FUNCTION_BLOCK FB_UnderfloorHeatingSystem EXTENDS FB_SystemContinous
VAR_INPUT
	bHeatingModeAutomatic : BOOL; //control mode: 0 = heating mode, 1 = cooling mode
	stAmbientState : ST_AmbientState;
END_VAR
VAR_OUTPUT
END_VAR
VAR
	{attribute 'OPC.UA.DA' := '1'}
	localSetParameters : ST_UnderfloorHeatingSetParameters;

	//default parameters
	localDefaultParameters : ST_UnderfloorHeatingDefaultParameters;	
	
	//pumps
	stPU425DefaultParameters : ST_PumpGrundfosMagna3DefaultParameters;
	PU425 : FB_PumpGrundfosMagna3 := (ST_DefaultParameters := stPU425DefaultParameters);	
	
	//valves
	stSV423DefaultParameters : ST_DiscreteValveDefaultParameters := (nFeedback := 3);
	stSV424DefaultParameters : ST_DiscreteValveDefaultParameters := (nFeedback := 3);
	stRV425DefaultParameters : ST_MixingValveDefaultParameters := (bFeedbackSignal := FALSE, tTaskCycleTime := GlobalVariables.tTaskCycleTime_MAIN, tCtrlCycleTime := GlobalVariables.tCtrlCycleTime_MAIN);	
	
	SV423 : FB_DiscreteValve := (ST_DefaultParameters := stSV423DefaultParameters); 
	SV424 : FB_DiscreteValve := (ST_DefaultParameters := stSV424DefaultParameters);
	RV425 : FB_MixingValve := (ST_DefaultParameters := stRV425DefaultParameters);
	
	//internal variables
	bHeatingMode 			: BOOL;
	bSetStatusOn_PU425 		: BOOL;
	bSetStatusOn_SV423		: BOOL;
	bSetStatusOn_SV424		: BOOL;
	bSetStatusOn_RV425 		: BOOL;
	fSetPoint_Internal 		: REAL;
	nControlMode_RV425 		: E_MixingValveControlMode; 	
	
	//characteristic curves and controllers
	CharacteristicCurve 			: FB_CTRL_FLOW_TEMP_SETPOINT_GEN;
	CharacteristicCurve_Parameters	: ST_CTRL_FLOW_TEMP_SETPOINT_GEN_PARAMS;
	
	//triggers
	SwitchToHeating : R_TRIG;
	SwitchToCooling : F_TRIG;
	bFinishedSwitchMode : BOOL := TRUE;
END_VAR

//check if heating mode has switched
SelectUnderfloorHeatingControlMode();
ControlUnderfloorHeating();
fSetPointAutomatic := fSetPoint_Internal;
SwitchToHeating(CLK := bHeatingMode);
SwitchToCooling(CLK := bHeatingMode);

//MAIN must be called before SwitchMode to prevent pump signal chattering (signal is written after SwitchMode function), SwitchMode may only be called if system is on
MAIN();

//disrupt calling SystemFlowControl via MAIN() when mode is switched and call SwitchMode()
IF ((SwitchToHeating.Q OR SwitchToCooling.Q) OR NOT bFinishedSwitchMode) AND bSetStatusOn THEN
	SwitchMode(bSwitchToHeating := bHeatingMode,
		bFinishedSwitchMode => bFinishedSwitchMode);
END_IF;

//pumps
PU425.GetState_Profibus();
PU425(bSetStatusOnAutomatic := bSetStatusOn_PU425,
	fSetPointAutomatic := 80,
	bAlgorithmPermission := bAlgorithmPermission,
	nControlModeAutomatic := 0);
PU425.SetState_Profibus();

//valves in thermal networks
RV425.GetState_AI();
RV425(bSetStatusOnAutomatic := bSetStatusOn_RV425,
	fSetPointAutomatic := fSetPoint_Internal,
	bAlgorithmPermission := bAlgorithmPermission,
	fTemperatureExternal := PU425.fTemperatureInternal,
	nControlModeAutomatic := nControlMode_RV425);
RV425.SetState_AO();

SV423.GetState_BI();
SV423(bSetStatusOnAutomatic := bSetStatusOn_SV423,
	bAlgorithmPermission := bAlgorithmPermission);
SV423.SetState_BO();

SV424.GetState_BI();
SV424(bSetStatusOnAutomatic := bSetStatusOn_SV423,
	bAlgorithmPermission := bAlgorithmPermission);
SV424.SetState_BO();

METHOD PROTECTED  CheckError : BOOL
VAR_INPUT
END_VAR
VAR_OUTPUT
	bError : BOOL;
END_VAR
VAR
END_VAR
//check pumps for errors
bError :=  PU425.bError;
END_METHOD

METHOD PRIVATE ControlUnderfloorHeating : BOOL
VAR_INPUT
END_VAR
VAR
END_VAR
CharacteristicCurve_Parameters.fAmbientTempMax := localDefaultParameters.aLimitsAmbientTemperature[2];
CharacteristicCurve_Parameters.fAmbientTempMin := localDefaultParameters.aLimitsAmbientTemperature[1];
CharacteristicCurve_Parameters.fForeRunTempMax := localDefaultParameters.aLimitsFeedTemperature[1];
CharacteristicCurve_Parameters.fForeRunTempMin := localDefaultParameters.aLimitsFeedTemperature[2];
CharacteristicCurve_Parameters.tCtrlCycleTime := GlobalVariables.tCtrlCycleTime_MAIN;
CharacteristicCurve_Parameters.tTaskCycleTime := GlobalVariables.tTaskCycleTime_MAIN;

CharacteristicCurve(fAmbientTemperature := stAmbientState.fOutsideTemperature,
	fOffsetTemperature := 0,
	bLimitFlowTemp := TRUE,
	stParams := CharacteristicCurve_Parameters);
fSetPoint_Internal := LREAL_TO_REAL(CharacteristicCurve.fOut);
	
IF bHeatingMode THEN
	nControlMode_RV425 := 1;
ELSE
	nControlMode_RV425 := 2;	
END_IF
END_METHOD

METHOD PROTECTED  Operational : BOOL
VAR_INPUT
END_VAR
VAR_OUTPUT
	bSwitchToWorking : BOOL := FALSE;
END_VAR
bSetStatusOn_RV425 := TRUE;
bSetStatusOn_PU425 := TRUE;

IF PU425.bStatusOn THEN
	bSwitchToWorking := TRUE;
END_IF
END_METHOD

METHOD PROTECTED  RampDown : BOOL
VAR_INPUT
END_VAR
VAR_OUTPUT
	bRampDownFinished : BOOL := FALSE;
END_VAR
bSetStatusOn_PU425 := FALSE;
bSetStatusOn_RV425 := FALSE;
bSetStatusOn_SV423 := FALSE;
bSetStatusOn_SV424 := FALSE;
	
IF SV423.localState.nPosition=3 AND SV424.localState.nPosition=3 THEN
	bRampDownFinished := TRUE;		
END_IF
END_METHOD

METHOD PROTECTED  RampUp : BOOL
VAR_INPUT
END_VAR
VAR_OUTPUT
	bRampUpFinished : BOOL := FALSE;
END_VAR
IF bHeatingMode THEN
	bSetStatusOn_SV423 := FALSE;
	bSetStatusOn_SV424 := FALSE;
	IF SV423.localState.nPosition=3 AND SV424.localState.nPosition=3 THEN
		bRampUpFinished := TRUE;		
	END_IF	
ELSE
	bSetStatusOn_SV423 := TRUE;
	bSetStatusOn_SV424 := TRUE;
	IF SV423.localState.nPosition=2 AND SV424.localState.nPosition=2 THEN
		bRampUpFinished := TRUE;		
	END_IF	
END_IF
END_METHOD

METHOD PRIVATE SelectUnderfloorHeatingControlMode : BOOL
VAR_INPUT
END_VAR
IF control.bManualModeActivated THEN
	bHeatingMode := localSetParameters.bHeatingModeManual;
ELSIF control.bAlgorithmModeActivated AND bAlgorithmPermission THEN
	bHeatingMode := localSetParameters.bHeatingModeAlgorithm;
ELSE
	bHeatingMode := bHeatingModeAutomatic;
END_IF
END_METHOD

METHOD PROTECTED   SetSetPointLimits : BOOL
VAR_INPUT
END_VAR
aSetPointLimits[1] := localDefaultParameters.aSetPointLimitsTemperature[1];
aSetPointLimits[2] := localDefaultParameters.aSetPointLimitsTemperature[2];
END_METHOD

METHOD PROTECTED  SetState : BOOL
VAR_INPUT
END_VAR
VAR_OUTPUT
END_VAR
fOperatingPoint := PU425.fTemperatureInternal;

controlState.bStatusOn := bSetStatusOn;
setPointState.aSetPointLimits := aSetPointLimits;
setPointState.fSetPoint := fSetPoint;
setPointState.fOperatingPoint := fOperatingPoint;
setPointState.sSetPointUnit := 'degreeC';
setPointState.sOperatingPointUnit := 'degreeC';
END_METHOD

METHOD PRIVATE SwitchMode : BOOL
VAR_INPUT
	bSwitchToHeating : BOOL; //if false switch to cooling
END_VAR
VAR_OUTPUT
	bFinishedSwitchMode : BOOL := FALSE;
END_VAR
VAR_INST
	bRampDownFinished : BOOL := FALSE;
END_VAR
//check system state
IF bRampDownFinished THEN
	IF bSwitchToHeating THEN
		//false - valve connects heating network
		bSetStatusOn_SV423 := TRUE;
		bSetStatusOn_SV424 := TRUE;	

		IF SV423.localState.nPosition=2 AND SV424.localState.nPosition=2 THEN
			//reset instant variable and switch on pump
			bRampDownFinished := FALSE;			
			bFinishedSwitchMode := TRUE;
			bSetStatusOn_PU425 := TRUE;
		END_IF
		
	ELSE
		//true - connects cooling network
		bSetStatusOn_SV423 := FALSE;
		bSetStatusOn_SV424 := FALSE;	

		IF SV423.localState.nPosition=3 AND SV424.localState.nPosition=3 THEN
			//reset instant variable and switch on pump
			bRampDownFinished := FALSE;			
			bFinishedSwitchMode := TRUE;
			bSetStatusOn_PU425 := TRUE;
		END_IF
	END_IF
ELSE
	bSetStatusOn_PU425 := FALSE;
	IF NOT PU425.bStatusOn THEN
		bRampDownFinished := TRUE;
	END_IF
END_IF
END_METHOD

METHOD PROTECTED  Working : BOOL
VAR_INPUT
END_VAR
VAR_OUTPUT
	bSwitchToOperational : BOOL := FALSE;
END_VAR
//empty method
END_METHOD

END_FUNCTION_BLOCK

(* stored: Version 1.1.0.1, ProductVersion 3.1.4024.10
   POU FB_UnderfloorHeatingSystem: Id {4efa52ab-487d-4cce-a8ee-6c4090219ec6}, SpecialFunc None
   Method CheckError: Id {b9b5fe8e-e7ff-4396-9357-ddff10f773aa}
   Method ControlUnderfloorHeating: Id {33d239a8-7df3-480e-902e-e6461385ded3}
   Method Operational: Id {b3659eec-c263-4bae-bfc6-63fd4bfd8556}
   Method RampDown: Id {9173a3c4-04c3-4530-96c4-77af03b435f0}
   Method RampUp: Id {ed258e40-1b81-4df7-9768-c25938f5bb5f}
   Method SelectUnderfloorHeatingControlMode: Id {7be6bcd7-4518-40f0-81a5-7bb610014654}
   Method SetSetPointLimits: Id {7a91eedd-ad13-4b09-b075-bc9157871f45}
   Method SetState: Id {5e916aa9-de43-48ca-bf50-12137a9ce652}
   Method SwitchMode: Id {db0b0ee2-1b40-45b2-95bd-b1cb07d07506}
   Method Working: Id {7c525aa6-95b6-42f5-b5b1-3574bb70abb3} *)
